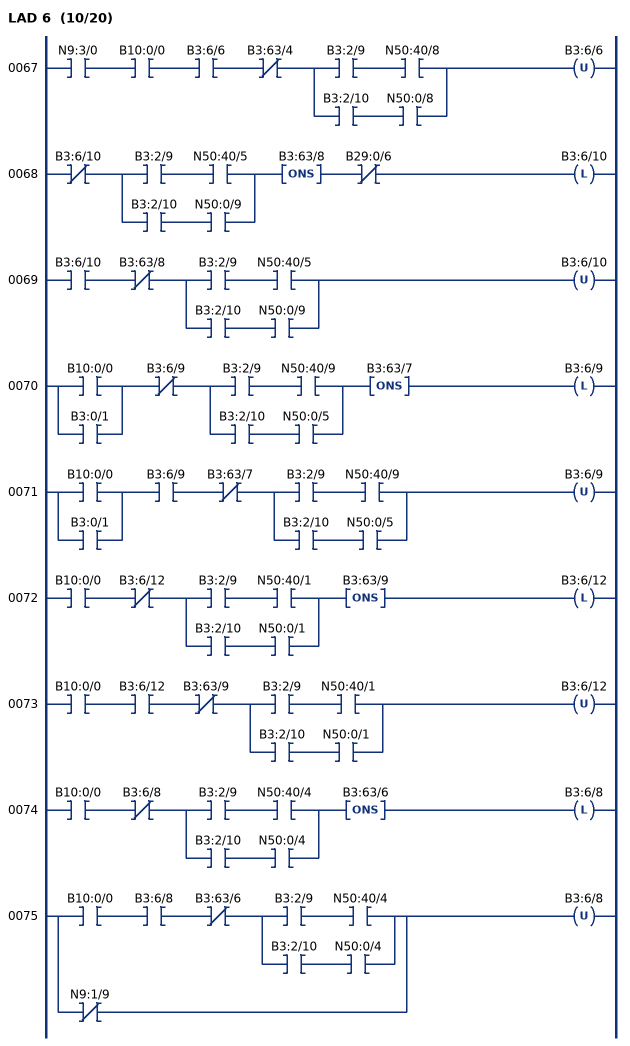
% Rung: 67 %
SOR XIC N9:3/0 XIC B10:0/0 XIC B3:6/6 XIO B3:63/4 BST XIC B3:2/9 XIC N50:40/8 NXB XIC B3:2/10 XIC N50:0/8 BND OTU B3:6/6 EOR
% Rung: 68 %
SOR XIO B3:6/10 BST XIC B3:2/9 XIC N50:40/5 NXB XIC B3:2/10 XIC N50:0/9 BND OSR B3:63/8 XIO B29:0/6 OTL B3:6/10 EOR
% Rung: 69 %
SOR XIC B3:6/10 XIO B3:63/8 BST XIC B3:2/9 XIC N50:40/5 NXB XIC B3:2/10 XIC N50:0/9 BND OTU B3:6/10 EOR
% Rung: 70 %
SOR BST XIC B10:0/0 NXB XIC B3:0/1 BND XIO B3:6/9 BST XIC B3:2/9 XIC N50:40/9 NXB XIC B3:2/10 XIC N50:0/5 BND OSR B3:63/7 OTL B3:6/9 EOR
% Rung: 71 %
SOR BST XIC B10:0/0 NXB XIC B3:0/1 BND XIC B3:6/9 XIO B3:63/7 BST XIC B3:2/9 XIC N50:40/9 NXB XIC B3:2/10 XIC N50:0/5 BND OTU B3:6/9 EOR
% Rung: 72 %
SOR XIC B10:0/0 XIO B3:6/12 BST XIC B3:2/9 XIC N50:40/1 NXB XIC B3:2/10 XIC N50:0/1 BND OSR B3:63/9 OTL B3:6/12 EOR
% Rung: 73 %
SOR XIC B10:0/0 XIC B3:6/12 XIO B3:63/9 BST XIC B3:2/9 XIC N50:40/1 NXB XIC B3:2/10 XIC N50:0/1 BND OTU B3:6/12 EOR
% Rung: 74 %
SOR XIC B10:0/0 XIO B3:6/8 BST XIC B3:2/9 XIC N50:40/4 NXB XIC B3:2/10 XIC N50:0/4 BND OSR B3:63/6 OTL B3:6/8 EOR
% Rung: 75 %
SOR BST XIC B10:0/0 XIC B3:6/8 XIO B3:63/6 BST XIC B3:2/9 XIC N50:40/4 NXB XIC B3:2/10 XIC N50:0/4 BND NXB XIO N9:1/9 BND OTU B3:6/8 EOR

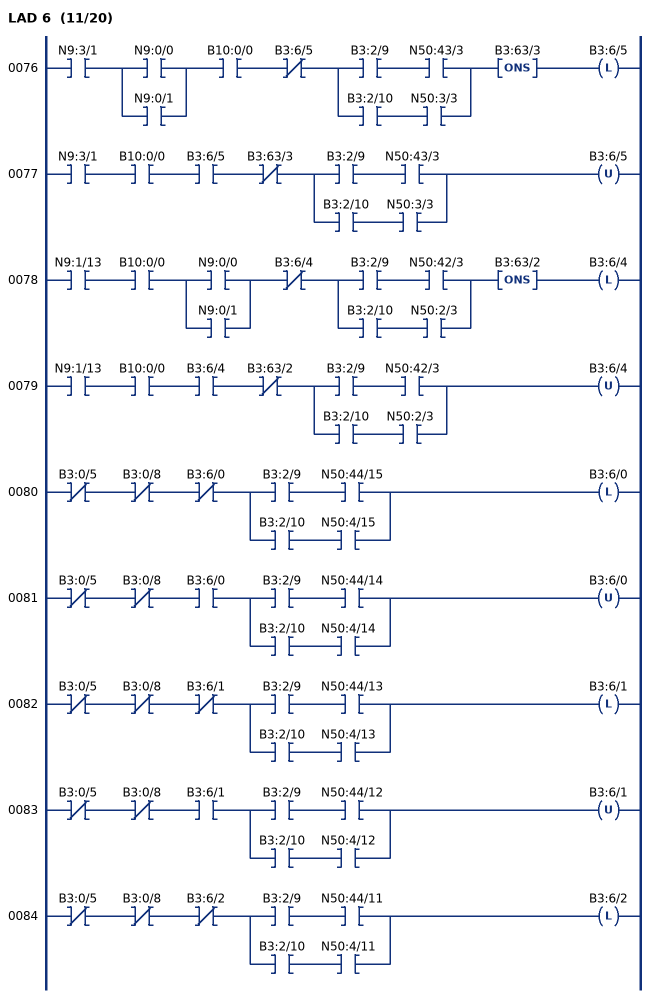
% Rung: 76 %
SOR XIC N9:3/1 BST XIC N9:0/0 NXB XIC N9:0/1 BND XIC B10:0/0 XIO B3:6/5 BST XIC B3:2/9 XIC N50:43/3 NXB XIC B3:2/10 XIC N50:3/3 BND OSR B3:63/3 OTL B3:6/5 EOR
% Rung: 77 %
SOR XIC N9:3/1 XIC B10:0/0 XIC B3:6/5 XIO B3:63/3 BST XIC B3:2/9 XIC N50:43/3 NXB XIC B3:2/10 XIC N50:3/3 BND OTU B3:6/5 EOR
% Rung: 78 %
SOR XIC N9:1/13 XIC B10:0/0 BST XIC N9:0/0 NXB XIC N9:0/1 BND XIO B3:6/4 BST XIC B3:2/9 XIC N50:42/3 NXB XIC B3:2/10 XIC N50:2/3 BND OSR B3:63/2 OTL B3:6/4 EOR
% Rung: 79 %
SOR XIC N9:1/13 XIC B10:0/0 XIC B3:6/4 XIO B3:63/2 BST XIC B3:2/9 XIC N50:42/3 NXB XIC B3:2/10 XIC N50:2/3 BND OTU B3:6/4 EOR
% Rung: 80 %
SOR XIO B3:0/5 XIO B3:0/8 XIO B3:6/0 BST XIC B3:2/9 XIC N50:44/15 NXB XIC B3:2/10 XIC N50:4/15 BND OTL B3:6/0 EOR
% Rung: 81 %
SOR XIO B3:0/5 XIO B3:0/8 XIC B3:6/0 BST XIC B3:2/9 XIC N50:44/14 NXB XIC B3:2/10 XIC N50:4/14 BND OTU B3:6/0 EOR
% Rung: 82 %
SOR XIO B3:0/5 XIO B3:0/8 XIO B3:6/1 BST XIC B3:2/9 XIC N50:44/13 NXB XIC B3:2/10 XIC N50:4/13 BND OTL B3:6/1 EOR
% Rung: 83 %
SOR XIO B3:0/5 XIO B3:0/8 XIC B3:6/1 BST XIC B3:2/9 XIC N50:44/12 NXB XIC B3:2/10 XIC N50:4/12 BND OTU B3:6/1 EOR
% Rung: 84 %
SOR XIO B3:0/5 XIO B3:0/8 XIO B3:6/2 BST XIC B3:2/9 XIC N50:44/11 NXB XIC B3:2/10 XIC N50:4/11 BND OTL B3:6/2 EOR

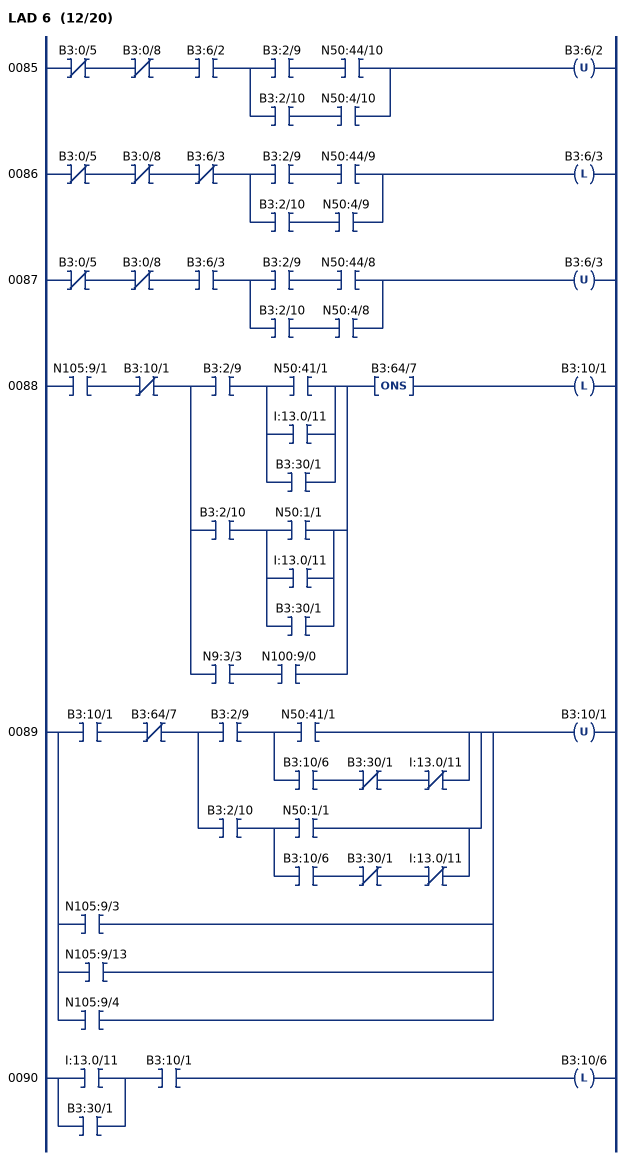
% Rung: 85 %
SOR XIO B3:0/5 XIO B3:0/8 XIC B3:6/2 BST XIC B3:2/9 XIC N50:44/10 NXB XIC B3:2/10 XIC N50:4/10 BND OTU B3:6/2 EOR
% Rung: 86 %
SOR XIO B3:0/5 XIO B3:0/8 XIO B3:6/3 BST XIC B3:2/9 XIC N50:44/9 NXB XIC B3:2/10 XIC N50:4/9 BND OTL B3:6/3 EOR
% Rung: 87 %
SOR XIO B3:0/5 XIO B3:0/8 XIC B3:6/3 BST XIC B3:2/9 XIC N50:44/8 NXB XIC B3:2/10 XIC N50:4/8 BND OTU B3:6/3 EOR
% Rung: 88 %
SOR XIC N105:9/1 XIO B3:10/1 BST XIC B3:2/9 BST XIC N50:41/1 NXB XIC I:13.0/11 NXB XIC B3:30/1 BND NXB XIC B3:2/10 BST XIC N50:1/1 NXB XIC I:13.0/11 NXB XIC B3:30/1 BND NXB XIC N9:3/3 XIC N100:9/0 BND OSR B3:64/7 OTL B3:10/1 EOR
% Rung: 89 %
SOR BST XIC B3:10/1 XIO B3:64/7 BST XIC B3:2/9 BST XIC N50:41/1 NXB XIC B3:10/6 XIO B3:30/1 XIO I:13.0/11 BND NXB XIC B3:2/10 BST XIC N50:1/1 NXB XIC B3:10/6 XIO B3:30/1 XIO I:13.0/11 BND BND NXB XIC N105:9/3 NXB XIC N105:9/13 NXB XIC N105:9/4 BND OTU B3:10/1 EOR
% Rung: 90 %
SOR BST XIC I:13.0/11 NXB XIC B3:30/1 BND XIC B3:10/1 OTL B3:10/6 EOR

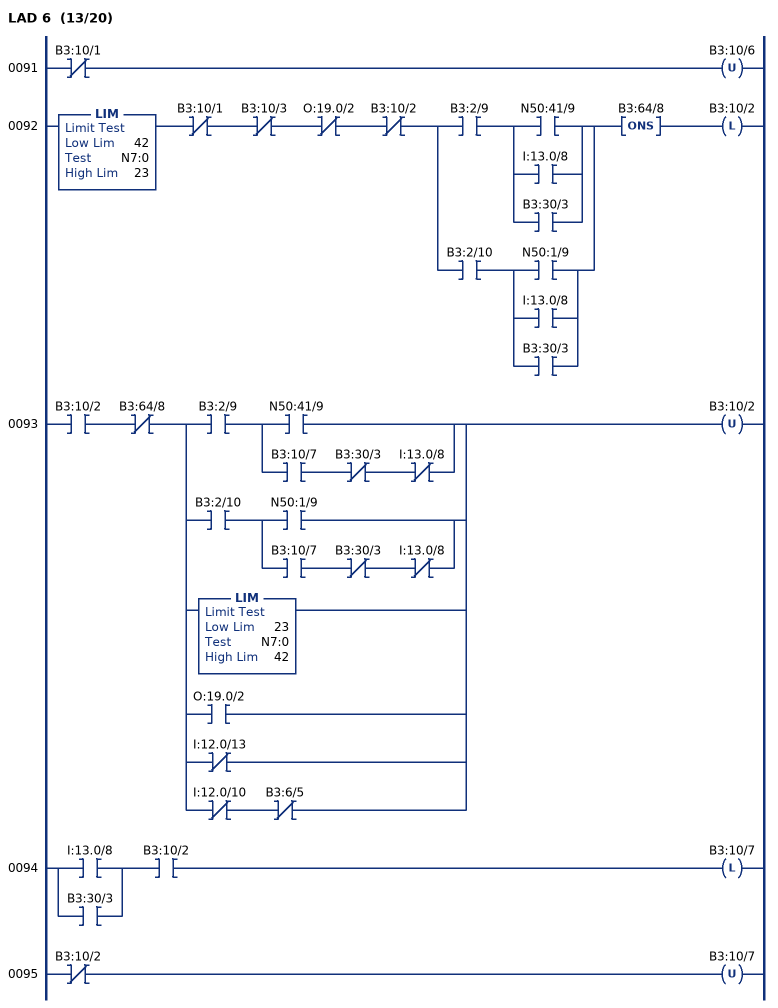
% Rung: 91 %
SOR XIO B3:10/1 OTU B3:10/6 EOR
% Rung: 92 %
SOR LIM 42 N7:0 23 XIO B3:10/1 XIO B3:10/3 XIO O:19.0/2 XIO B3:10/2 BST XIC B3:2/9 BST XIC N50:41/9 NXB XIC I:13.0/8 NXB XIC B3:30/3 BND NXB XIC B3:2/10 BST XIC N50:1/9 NXB XIC I:13.0/8 NXB XIC B3:30/3 BND BND OSR B3:64/8 OTL B3:10/2 EOR
% Rung: 93 %
SOR XIC B3:10/2 XIO B3:64/8 BST XIC B3:2/9 BST XIC N50:41/9 NXB XIC B3:10/7 XIO B3:30/3 XIO I:13.0/8 BND NXB XIC B3:2/10 BST XIC N50:1/9 NXB XIC B3:10/7 XIO B3:30/3 XIO I:13.0/8 BND NXB LIM 23 N7:0 42 NXB XIC O:19.0/2 NXB XIO I:12.0/13 NXB XIO I:12.0/10 XIO B3:6/5 BND OTU B3:10/2 EOR
% Rung: 94 %
SOR BST XIC I:13.0/8 NXB XIC B3:30/3 BND XIC B3:10/2 OTL B3:10/7 EOR
% Rung: 95 %
SOR XIO B3:10/2 OTU B3:10/7 EOR

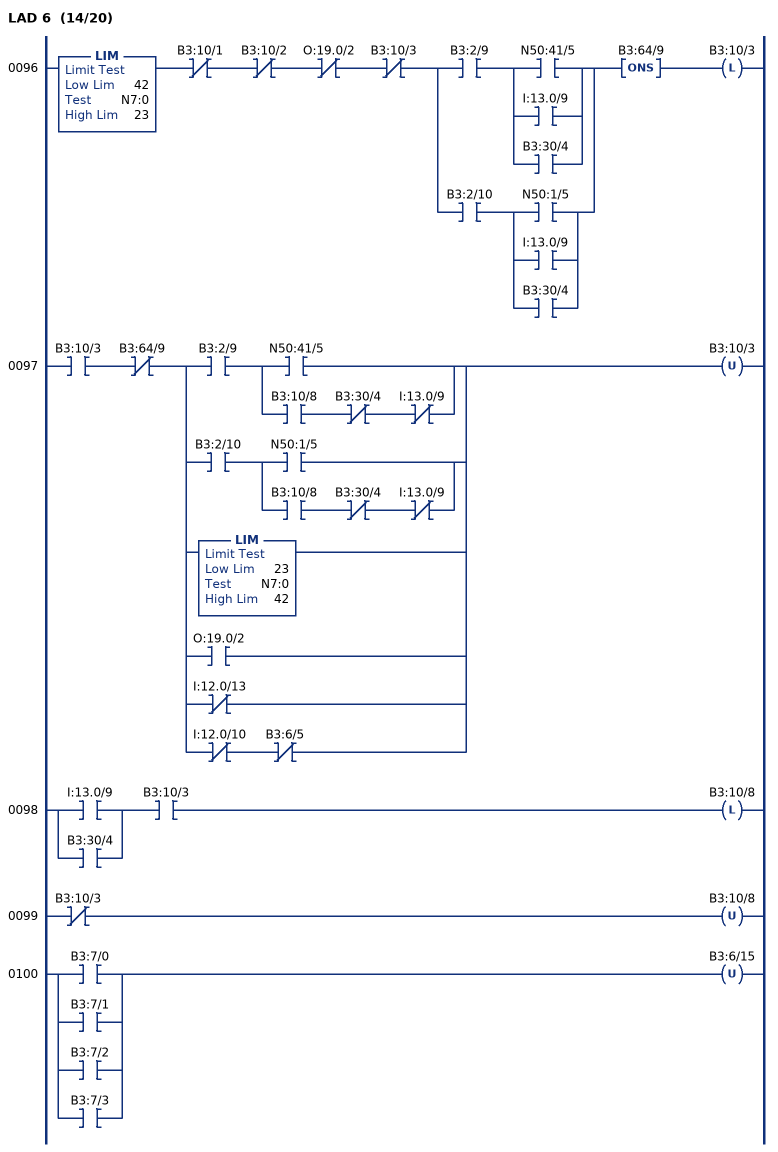
% Rung: 96 %
SOR LIM 42 N7:0 23 XIO B3:10/1 XIO B3:10/2 XIO O:19.0/2 XIO B3:10/3 BST XIC B3:2/9 BST XIC N50:41/5 NXB XIC I:13.0/9 NXB XIC B3:30/4 BND NXB XIC B3:2/10 BST XIC N50:1/5 NXB XIC I:13.0/9 NXB XIC B3:30/4 BND BND OSR B3:64/9 OTL B3:10/3 EOR
% Rung: 97 %
SOR XIC B3:10/3 XIO B3:64/9 BST XIC B3:2/9 BST XIC N50:41/5 NXB XIC B3:10/8 XIO B3:30/4 XIO I:13.0/9 BND NXB XIC B3:2/10 BST XIC N50:1/5 NXB XIC B3:10/8 XIO B3:30/4 XIO I:13.0/9 BND NXB LIM 23 N7:0 42 NXB XIC O:19.0/2 NXB XIO I:12.0/13 NXB XIO I:12.0/10 XIO B3:6/5 BND OTU B3:10/3 EOR
% Rung: 98 %
SOR BST XIC I:13.0/9 NXB XIC B3:30/4 BND XIC B3:10/3 OTL B3:10/8 EOR
% Rung: 99 %
SOR XIO B3:10/3 OTU B3:10/8 EOR
% Rung: 100 %
SOR BST XIC B3:7/0 NXB XIC B3:7/1 NXB XIC B3:7/2 NXB XIC B3:7/3 BND OTU B3:6/15 EOR

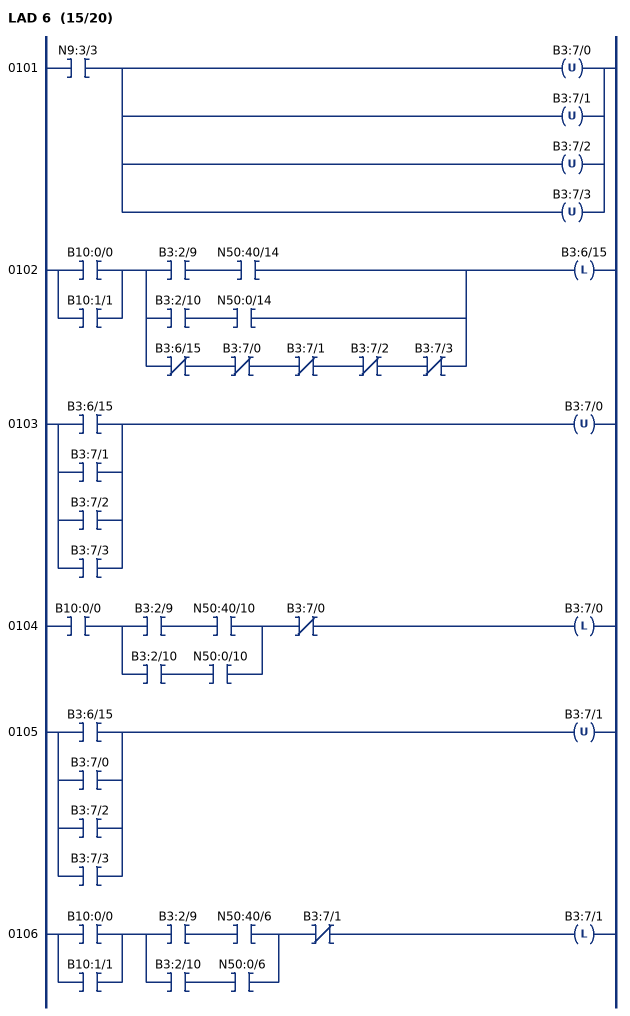
% Rung: 101 %
SOR XIC N9:3/3 BST OTU B3:7/0 NXB OTU B3:7/1 NXB OTU B3:7/2 NXB OTU B3:7/3 BND EOR
% Rung: 102 %
SOR BST XIC B10:0/0 NXB XIC B10:1/1 BND BST XIC B3:2/9 XIC N50:40/14 NXB XIC B3:2/10 XIC N50:0/14 NXB XIO B3:6/15 XIO B3:7/0 XIO B3:7/1 XIO B3:7/2 XIO B3:7/3 BND OTL B3:6/15 EOR
% Rung: 103 %
SOR BST XIC B3:6/15 NXB XIC B3:7/1 NXB XIC B3:7/2 NXB XIC B3:7/3 BND OTU B3:7/0 EOR
% Rung: 104 %
SOR XIC B10:0/0 BST XIC B3:2/9 XIC N50:40/10 NXB XIC B3:2/10 XIC N50:0/10 BND XIO B3:7/0 OTL B3:7/0 EOR
% Rung: 105 %
SOR BST XIC B3:6/15 NXB XIC B3:7/0 NXB XIC B3:7/2 NXB XIC B3:7/3 BND OTU B3:7/1 EOR
% Rung: 106 %
SOR BST XIC B10:0/0 NXB XIC B10:1/1 BND BST XIC B3:2/9 XIC N50:40/6 NXB XIC B3:2/10 XIC N50:0/6 BND XIO B3:7/1 OTL B3:7/1 EOR

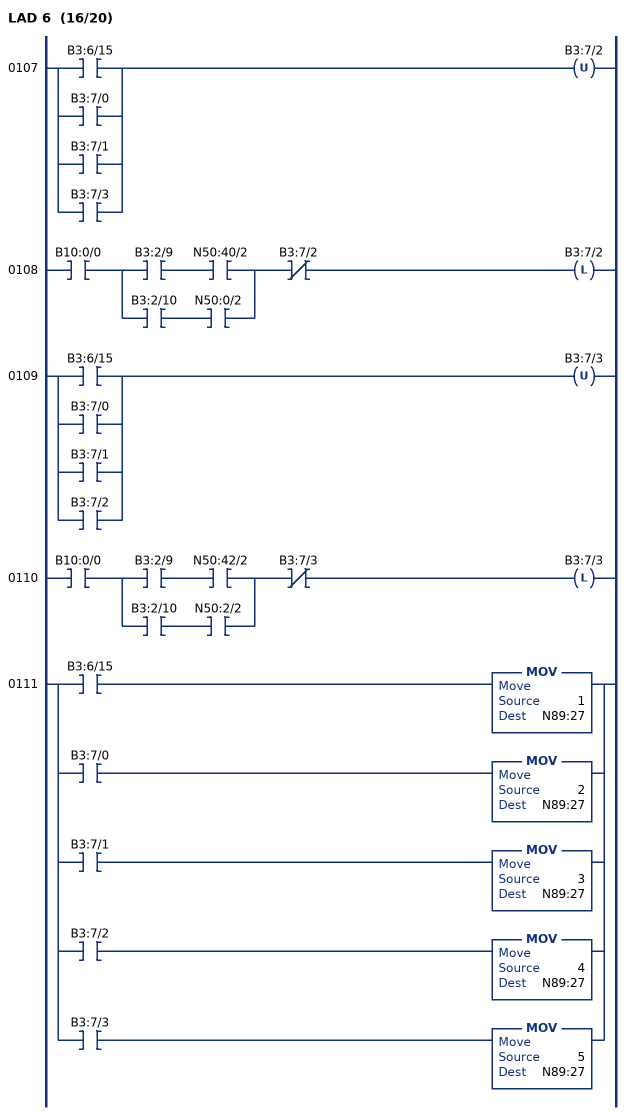
% Rung: 107 %
SOR BST XIC B3:6/15 NXB XIC B3:7/0 NXB XIC B3:7/1 NXB XIC B3:7/3 BND OTU B3:7/2 EOR
% Rung: 108 %
SOR XIC B10:0/0 BST XIC B3:2/9 XIC N50:40/2 NXB XIC B3:2/10 XIC N50:0/2 BND XIO B3:7/2 OTL B3:7/2 EOR
% Rung: 109 %
SOR BST XIC B3:6/15 NXB XIC B3:7/0 NXB XIC B3:7/1 NXB XIC B3:7/2 BND OTU B3:7/3 EOR
% Rung: 110 %
SOR XIC B10:0/0 BST XIC B3:2/9 XIC N50:42/2 NXB XIC B3:2/10 XIC N50:2/2 BND XIO B3:7/3 OTL B3:7/3 EOR
% Rung: 111 %
SOR BST XIC B3:6/15 MOV 1 N89:27 NXB XIC B3:7/0 MOV 2 N89:27 NXB XIC B3:7/1 MOV 3 N89:27 NXB XIC B3:7/2 MOV 4 N89:27 NXB XIC B3:7/3 MOV 5 N89:27 BND EOR

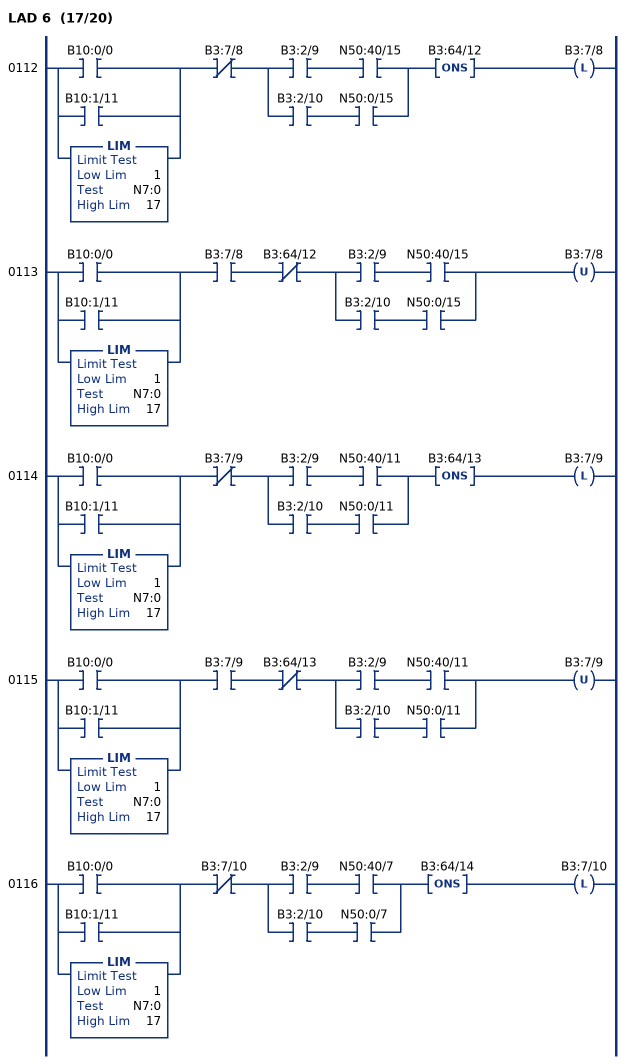
% Rung: 112 %
SOR BST XIC B10:0/0 NXB XIC B10:1/11 NXB LIM 1 N7:0 17 BND XIO B3:7/8 BST XIC B3:2/9 XIC N50:40/15 NXB XIC B3:2/10 XIC N50:0/15 BND OSR B3:64/12 OTL B3:7/8 EOR
% Rung: 113 %
SOR BST XIC B10:0/0 NXB XIC B10:1/11 NXB LIM 1 N7:0 17 BND XIC B3:7/8 XIO B3:64/12 BST XIC B3:2/9 XIC N50:40/15 NXB XIC B3:2/10 XIC N50:0/15 BND OTU B3:7/8 EOR
% Rung: 114 %
SOR BST XIC B10:0/0 NXB XIC B10:1/11 NXB LIM 1 N7:0 17 BND XIO B3:7/9 BST XIC B3:2/9 XIC N50:40/11 NXB XIC B3:2/10 XIC N50:0/11 BND OSR B3:64/13 OTL B3:7/9 EOR
% Rung: 115 %
SOR BST XIC B10:0/0 NXB XIC B10:1/11 NXB LIM 1 N7:0 17 BND XIC B3:7/9 XIO B3:64/13 BST XIC B3:2/9 XIC N50:40/11 NXB XIC B3:2/10 XIC N50:0/11 BND OTU B3:7/9 EOR
% Rung: 116 %
SOR BST XIC B10:0/0 NXB XIC B10:1/11 NXB LIM 1 N7:0 17 BND XIO B3:7/10 BST XIC B3:2/9 XIC N50:40/7 NXB XIC B3:2/10 XIC N50:0/7 BND OSR B3:64/14 OTL B3:7/10 EOR

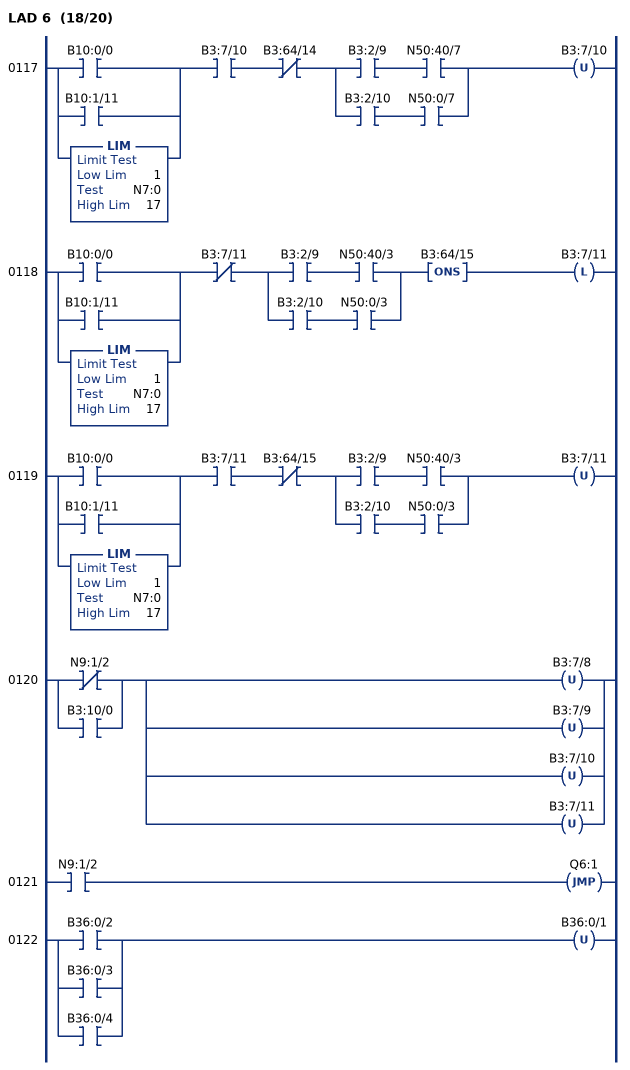
% Rung: 117 %
SOR BST XIC B10:0/0 NXB XIC B10:1/11 NXB LIM 1 N7:0 17 BND XIC B3:7/10 XIO B3:64/14 BST XIC B3:2/9 XIC N50:40/7 NXB XIC B3:2/10 XIC N50:0/7 BND OTU B3:7/10 EOR
% Rung: 118 %
SOR BST XIC B10:0/0 NXB XIC B10:1/11 NXB LIM 1 N7:0 17 BND XIO B3:7/11 BST XIC B3:2/9 XIC N50:40/3 NXB XIC B3:2/10 XIC N50:0/3 BND OSR B3:64/15 OTL B3:7/11 EOR
% Rung: 119 %
SOR BST XIC B10:0/0 NXB XIC B10:1/11 NXB LIM 1 N7:0 17 BND XIC B3:7/11 XIO B3:64/15 BST XIC B3:2/9 XIC N50:40/3 NXB XIC B3:2/10 XIC N50:0/3 BND OTU B3:7/11 EOR
% Rung: 120 %
SOR BST XIO N9:1/2 NXB XIC B3:10/0 BND BST OTU B3:7/8 NXB OTU B3:7/9 NXB OTU B3:7/10 NXB OTU B3:7/11 BND EOR
% Rung: 121 %
SOR XIC N9:1/2 JMP Q6:1 EOR
% Rung: 122 %
SOR BST XIC B36:0/2 NXB XIC B36:0/3 NXB XIC B36:0/4 BND OTU B36:0/1 EOR

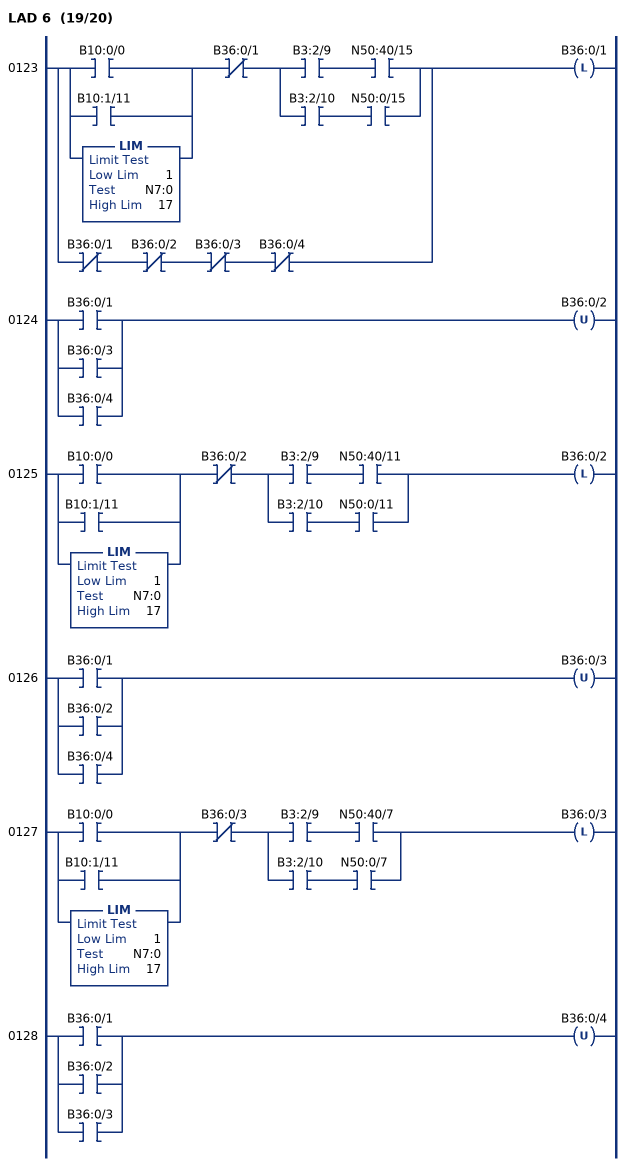
% Rung: 123 %
SOR BST BST XIC B10:0/0 NXB XIC B10:1/11 NXB LIM 1 N7:0 17 BND XIO B36:0/1 BST XIC B3:2/9 XIC N50:40/15 NXB XIC B3:2/10 XIC N50:0/15 BND NXB XIO B36:0/1 XIO B36:0/2 XIO B36:0/3 XIO B36:0/4 BND OTL B36:0/1 EOR
% Rung: 124 %
SOR BST XIC B36:0/1 NXB XIC B36:0/3 NXB XIC B36:0/4 BND OTU B36:0/2 EOR
% Rung: 125 %
SOR BST XIC B10:0/0 NXB XIC B10:1/11 NXB LIM 1 N7:0 17 BND XIO B36:0/2 BST XIC B3:2/9 XIC N50:40/11 NXB XIC B3:2/10 XIC N50:0/11 BND OTL B36:0/2 EOR
% Rung: 126 %
SOR BST XIC B36:0/1 NXB XIC B36:0/2 NXB XIC B36:0/4 BND OTU B36:0/3 EOR
% Rung: 127 %
SOR BST XIC B10:0/0 NXB XIC B10:1/11 NXB LIM 1 N7:0 17 BND XIO B36:0/3 BST XIC B3:2/9 XIC N50:40/7 NXB XIC B3:2/10 XIC N50:0/7 BND OTL B36:0/3 EOR
% Rung: 128 %
SOR BST XIC B36:0/1 NXB XIC B36:0/2 NXB XIC B36:0/3 BND OTU B36:0/4 EOR

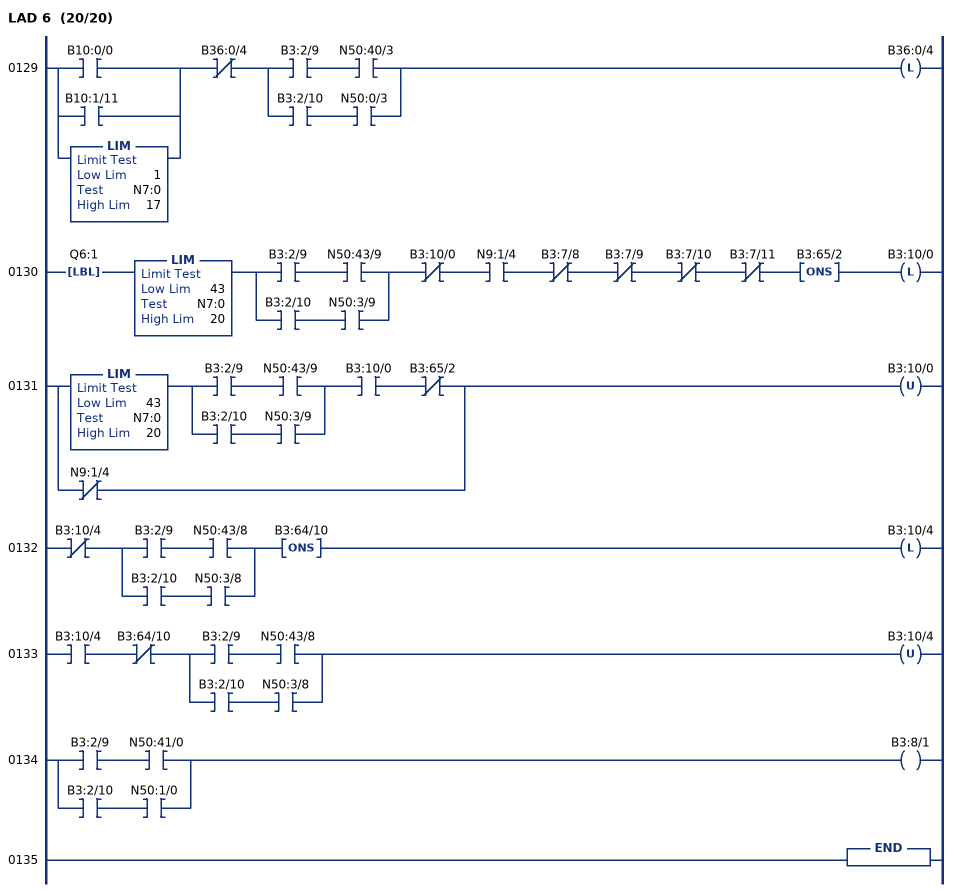
% Rung: 129 %
SOR BST XIC B10:0/0 NXB XIC B10:1/11 NXB LIM 1 N7:0 17 BND XIO B36:0/4 BST XIC B3:2/9 XIC N50:40/3 NXB XIC B3:2/10 XIC N50:0/3 BND OTL B36:0/4 EOR
% Rung: 130 %
SOR LBL Q6:1 LIM 43 N7:0 20 BST XIC B3:2/9 XIC N50:43/9 NXB XIC B3:2/10 XIC N50:3/9 BND XIO B3:10/0 XIC N9:1/4 XIO B3:7/8 XIO B3:7/9 XIO B3:7/10 XIO B3:7/11 OSR B3:65/2 OTL B3:10/0 EOR
% Rung: 131 %
SOR BST LIM 43 N7:0 20 BST XIC B3:2/9 XIC N50:43/9 NXB XIC B3:2/10 XIC N50:3/9 BND XIC B3:10/0 XIO B3:65/2 NXB XIO N9:1/4 BND OTU B3:10/0 EOR
% Rung: 132 %
SOR XIO B3:10/4 BST XIC B3:2/9 XIC N50:43/8 NXB XIC B3:2/10 XIC N50:3/8 BND OSR B3:64/10 OTL B3:10/4 EOR
% Rung: 133 %
SOR XIC B3:10/4 XIO B3:64/10 BST XIC B3:2/9 XIC N50:43/8 NXB XIC B3:2/10 XIC N50:3/8 BND OTU B3:10/4 EOR
% Rung: 134 %
SOR BST XIC B3:2/9 XIC N50:41/0 NXB XIC B3:2/10 XIC N50:1/0 BND OTE B3:8/1 EOR
% Rung: 135 %
SOR END EOR

LADDER 9
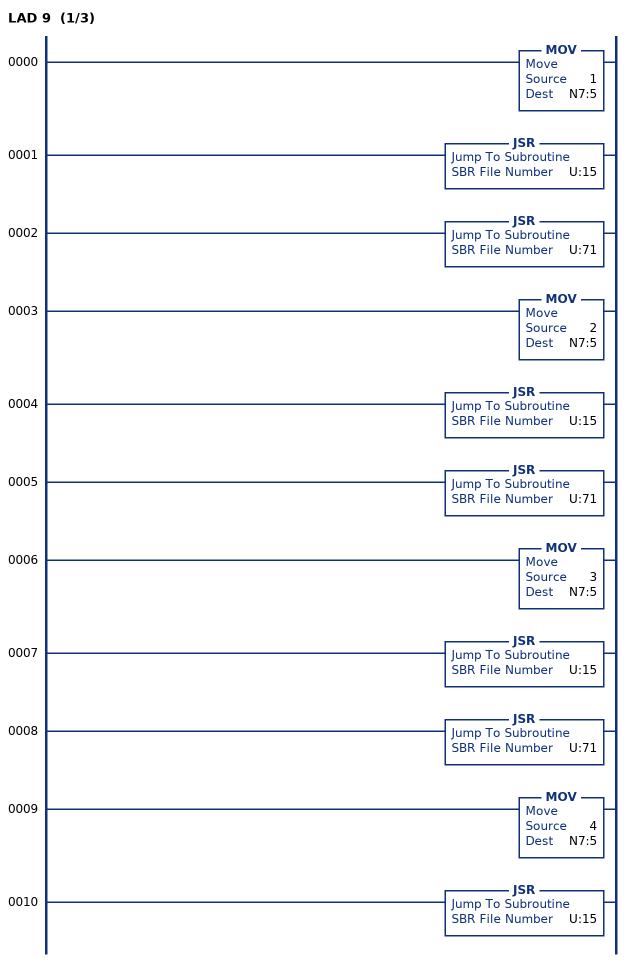
% Rung: 0 %
SOR MOV 1 N7:5 EOR
% Rung: 1 %
SOR JSR U:15 EOR
% Rung: 2 %
SOR JSR U:71 EOR
% Rung: 3 %
SOR MOV 2 N7:5 EOR
% Rung: 4 %
SOR JSR U:15 EOR
% Rung: 5 %
SOR JSR U:71 EOR
% Rung: 6 %
SOR MOV 3 N7:5 EOR
% Rung: 7 %
SOR JSR U:15 EOR
% Rung: 8 %
SOR JSR U:71 EOR
% Rung: 9 %
SOR MOV 4 N7:5 EOR
% Rung: 10 %
SOR JSR U:15 EOR

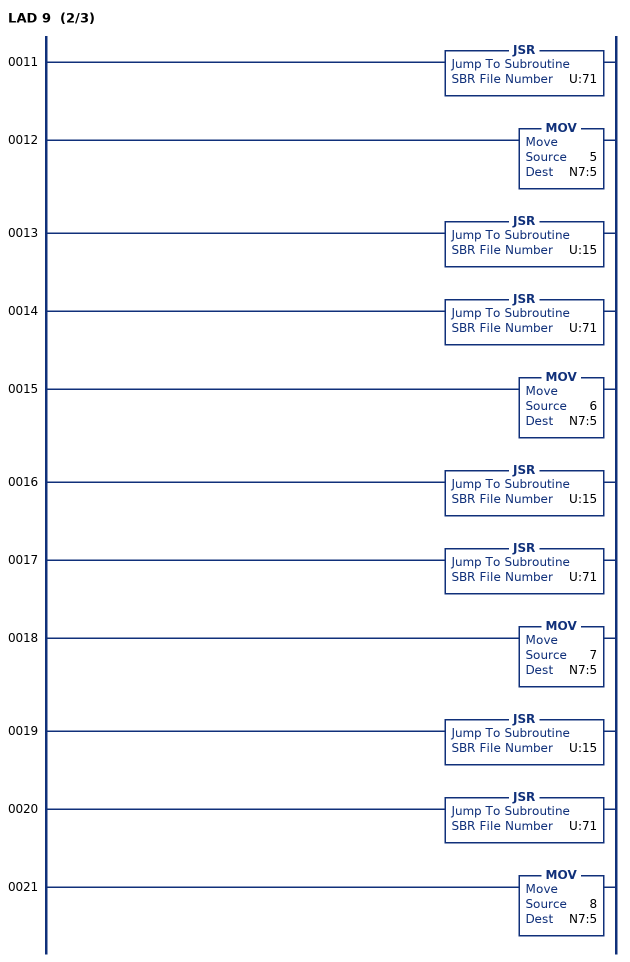
% Rung: 11 %
SOR JSR U:71 EOR
% Rung: 12 %
SOR MOV 5 N7:5 EOR
% Rung: 13 %
SOR JSR U:15 EOR
% Rung: 14 %
SOR JSR U:71 EOR
% Rung: 15 %
SOR MOV 6 N7:5 EOR
% Rung: 16 %
SOR JSR U:15 EOR
% Rung: 17 %
SOR JSR U:71 EOR
% Rung: 18 %
SOR MOV 7 N7:5 EOR
% Rung: 19 %
SOR JSR U:15 EOR
% Rung: 20 %
SOR JSR U:71 EOR
% Rung: 21 %
SOR MOV 8 N7:5 EOR

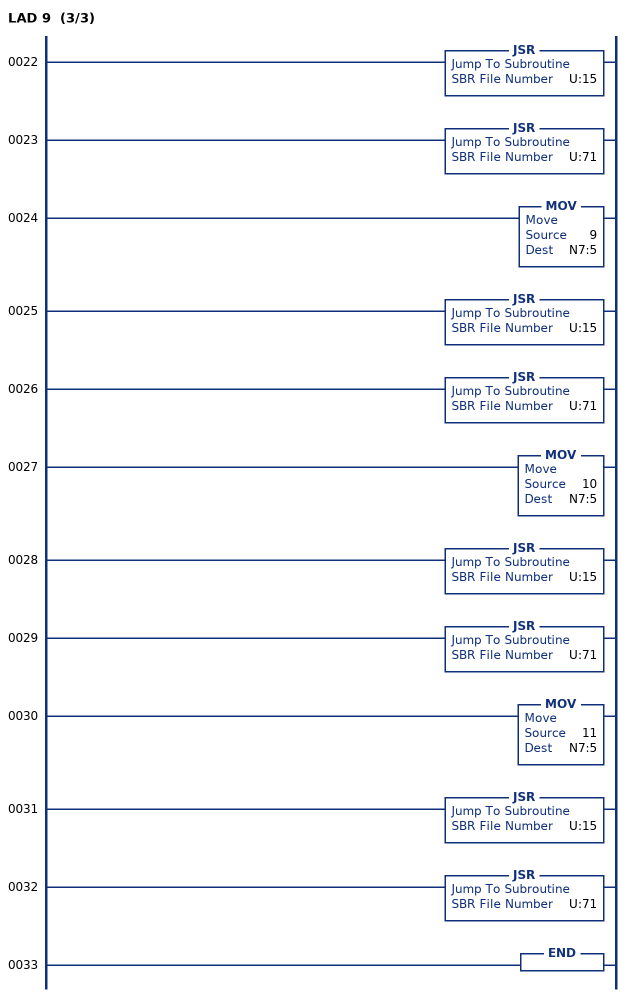
% Rung: 22 %
SOR JSR U:15 EOR
% Rung: 23 %
SOR JSR U:71 EOR
% Rung: 24 %
SOR MOV 9 N7:5 EOR
% Rung: 25 %
SOR JSR U:15 EOR
% Rung: 26 %
SOR JSR U:71 EOR
% Rung: 27 %
SOR MOV 10 N7:5 EOR
% Rung: 28 %
SOR JSR U:15 EOR
% Rung: 29 %
SOR JSR U:71 EOR
% Rung: 30 %
SOR MOV 11 N7:5 EOR
% Rung: 31 %
SOR JSR U:15 EOR
% Rung: 32 %
SOR JSR U:71 EOR
% Rung: 33 %
SOR END EOR

LADDER 10
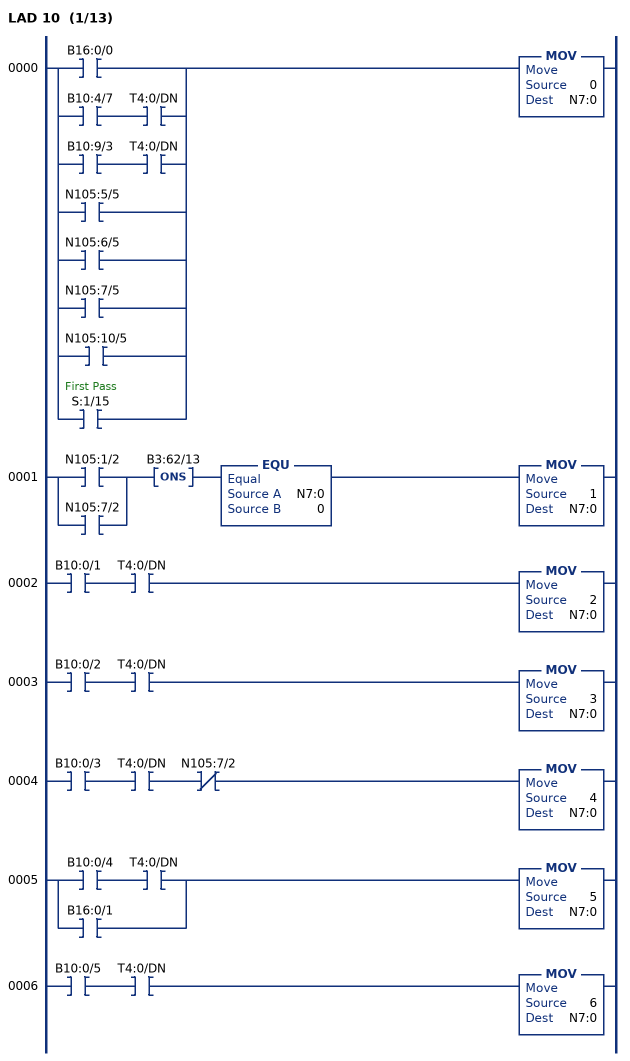
% Rung: 0 %
SOR BST XIC B16:0/0 NXB XIC B10:4/7 XIC T4:0/DN NXB XIC B10:9/3 XIC T4:0/DN NXB XIC N105:5/5 NXB XIC N105:6/5 NXB XIC N105:7/5 NXB XIC N105:10/5 NXB XIC S:1/15 BND MOV 0 N7:0 EOR
%   S:1/15  "First Pass" %
% Rung: 1 %
SOR BST XIC N105:1/2 NXB XIC N105:7/2 BND OSR B3:62/13 EQU N7:0 0 MOV 1 N7:0 EOR
% Rung: 2 %
SOR XIC B10:0/1 XIC T4:0/DN MOV 2 N7:0 EOR
% Rung: 3 %
SOR XIC B10:0/2 XIC T4:0/DN MOV 3 N7:0 EOR
% Rung: 4 %
SOR XIC B10:0/3 XIC T4:0/DN XIO N105:7/2 MOV 4 N7:0 EOR
% Rung: 5 %
SOR BST XIC B10:0/4 XIC T4:0/DN NXB XIC B16:0/1 BND MOV 5 N7:0 EOR
% Rung: 6 %
SOR XIC B10:0/5 XIC T4:0/DN MOV 6 N7:0 EOR

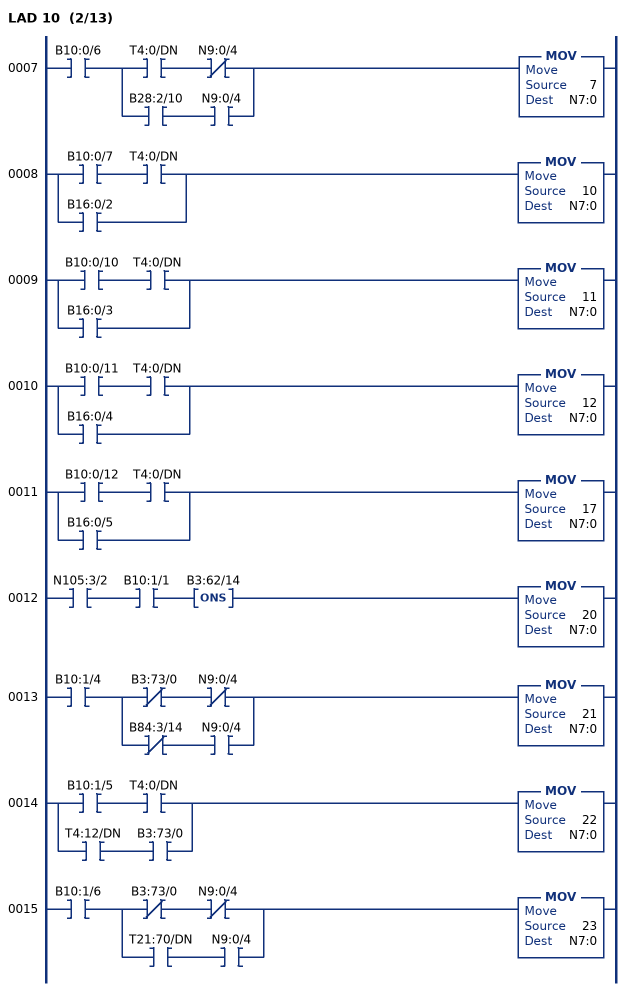
% Rung: 7 %
SOR XIC B10:0/6 BST XIC T4:0/DN XIO N9:0/4 NXB XIC B28:2/10 XIC N9:0/4 BND MOV 7 N7:0 EOR
% Rung: 8 %
SOR BST XIC B10:0/7 XIC T4:0/DN NXB XIC B16:0/2 BND MOV 10 N7:0 EOR
% Rung: 9 %
SOR BST XIC B10:0/10 XIC T4:0/DN NXB XIC B16:0/3 BND MOV 11 N7:0 EOR
% Rung: 10 %
SOR BST XIC B10:0/11 XIC T4:0/DN NXB XIC B16:0/4 BND MOV 12 N7:0 EOR
% Rung: 11 %
SOR BST XIC B10:0/12 XIC T4:0/DN NXB XIC B16:0/5 BND MOV 17 N7:0 EOR
% Rung: 12 %
SOR XIC N105:3/2 XIC B10:1/1 OSR B3:62/14 MOV 20 N7:0 EOR
% Rung: 13 %
SOR XIC B10:1/4 BST XIO B3:73/0 XIO N9:0/4 NXB XIO B84:3/14 XIC N9:0/4 BND MOV 21 N7:0 EOR
% Rung: 14 %
SOR BST XIC B10:1/5 XIC T4:0/DN NXB XIC T4:12/DN XIC B3:73/0 BND MOV 22 N7:0 EOR
% Rung: 15 %
SOR XIC B10:1/6 BST XIO B3:73/0 XIO N9:0/4 NXB XIC T21:70/DN XIC N9:0/4 BND MOV 23 N7:0 EOR

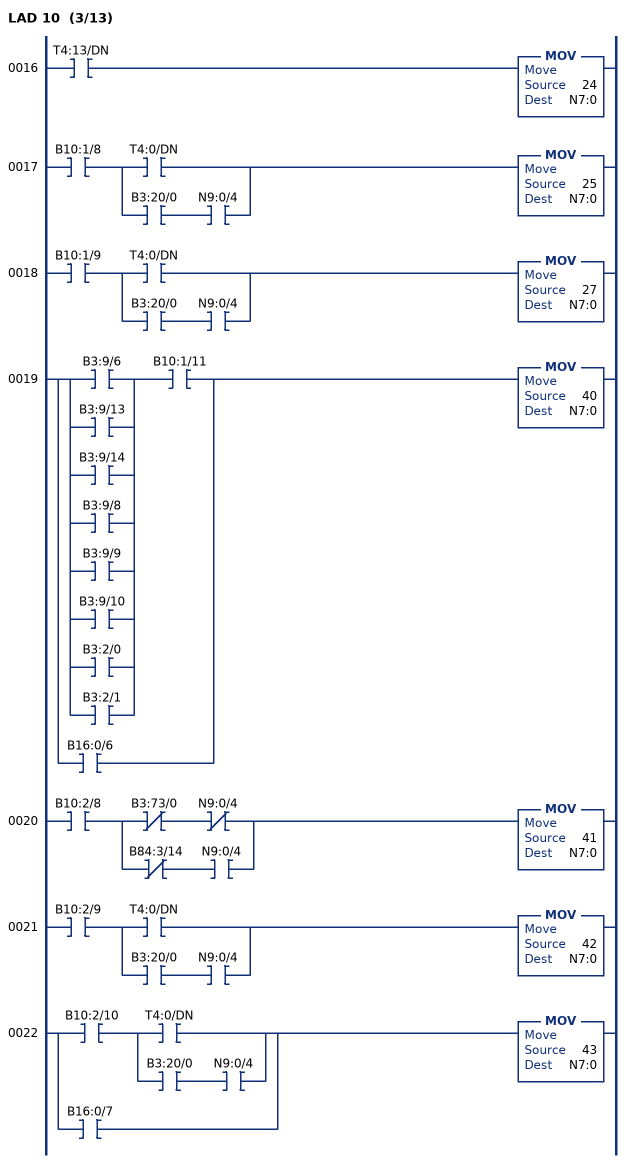
% Rung: 16 %
SOR XIC T4:13/DN MOV 24 N7:0 EOR
% Rung: 17 %
SOR XIC B10:1/8 BST XIC T4:0/DN NXB XIC B3:20/0 XIC N9:0/4 BND MOV 25 N7:0 EOR
% Rung: 18 %
SOR XIC B10:1/9 BST XIC T4:0/DN NXB XIC B3:20/0 XIC N9:0/4 BND MOV 27 N7:0 EOR
% Rung: 19 %
SOR BST BST XIC B3:9/6 NXB XIC B3:9/13 NXB XIC B3:9/14 NXB XIC B3:9/8 NXB XIC B3:9/9 NXB XIC B3:9/10 NXB XIC B3:2/0 NXB XIC B3:2/1 BND XIC B10:1/11 NXB XIC B16:0/6 BND MOV 40 N7:0 EOR
% Rung: 20 %
SOR XIC B10:2/8 BST XIO B3:73/0 XIO N9:0/4 NXB XIO B84:3/14 XIC N9:0/4 BND MOV 41 N7:0 EOR
% Rung: 21 %
SOR XIC B10:2/9 BST XIC T4:0/DN NXB XIC B3:20/0 XIC N9:0/4 BND MOV 42 N7:0 EOR
% Rung: 22 %
SOR BST XIC B10:2/10 BST XIC T4:0/DN NXB XIC B3:20/0 XIC N9:0/4 BND NXB XIC B16:0/7 BND MOV 43 N7:0 EOR

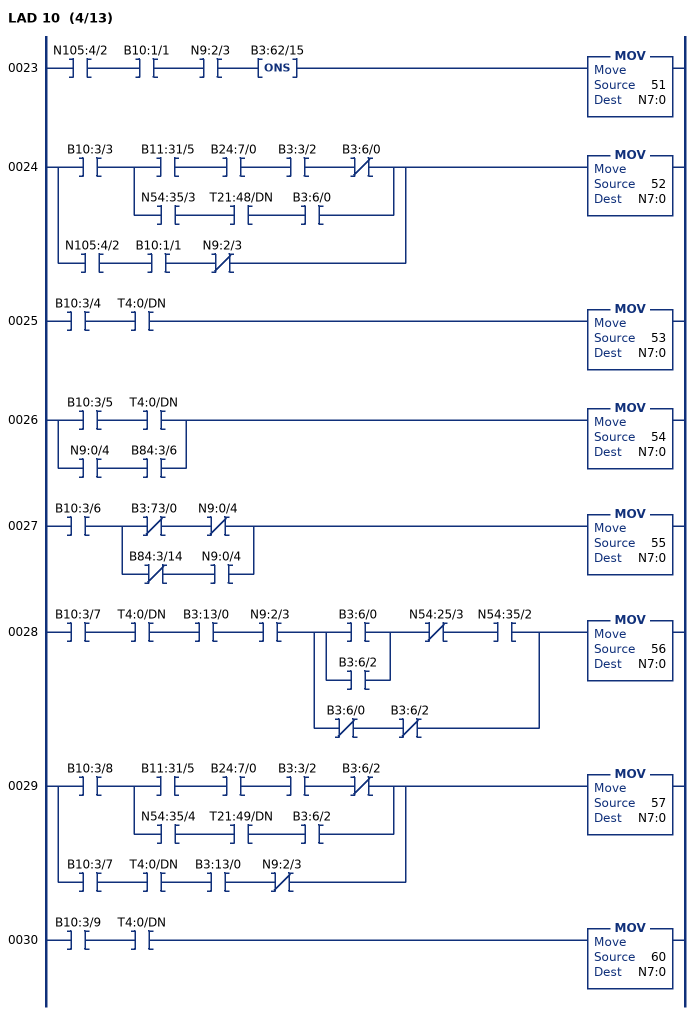
% Rung: 23 %
SOR XIC N105:4/2 XIC B10:1/1 XIC N9:2/3 OSR B3:62/15 MOV 51 N7:0 EOR
% Rung: 24 %
SOR BST XIC B10:3/3 BST XIC B11:31/5 XIC B24:7/0 XIC B3:3/2 XIO B3:6/0 NXB XIC N54:35/3 XIC T21:48/DN XIC B3:6/0 BND NXB XIC N105:4/2 XIC B10:1/1 XIO N9:2/3 BND MOV 52 N7:0 EOR
% Rung: 25 %
SOR XIC B10:3/4 XIC T4:0/DN MOV 53 N7:0 EOR
% Rung: 26 %
SOR BST XIC B10:3/5 XIC T4:0/DN NXB XIC N9:0/4 XIC B84:3/6 BND MOV 54 N7:0 EOR
% Rung: 27 %
SOR XIC B10:3/6 BST XIO B3:73/0 XIO N9:0/4 NXB XIO B84:3/14 XIC N9:0/4 BND MOV 55 N7:0 EOR
% Rung: 28 %
SOR XIC B10:3/7 XIC T4:0/DN XIC B3:13/0 XIC N9:2/3 BST BST XIC B3:6/0 NXB XIC B3:6/2 BND XIO N54:25/3 XIC N54:35/2 NXB XIO B3:6/0 XIO B3:6/2 BND MOV 56 N7:0 EOR
% Rung: 29 %
SOR BST XIC B10:3/8 BST XIC B11:31/5 XIC B24:7/0 XIC B3:3/2 XIO B3:6/2 NXB XIC N54:35/4 XIC T21:49/DN XIC B3:6/2 BND NXB XIC B10:3/7 XIC T4:0/DN XIC B3:13/0 XIO N9:2/3 BND MOV 57 N7:0 EOR
% Rung: 30 %
SOR XIC B10:3/9 XIC T4:0/DN MOV 60 N7:0 EOR

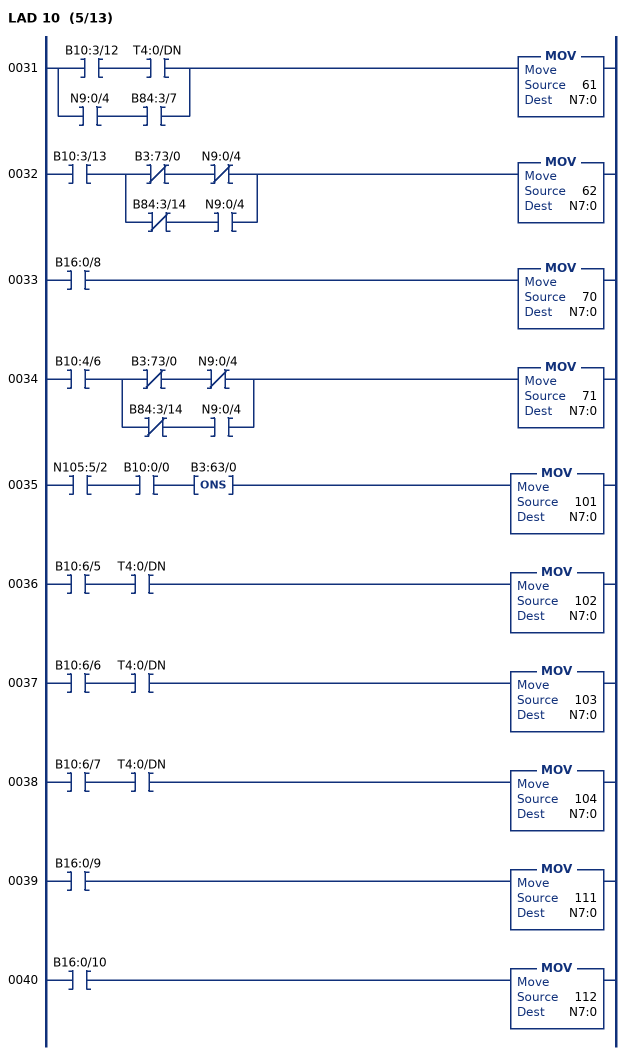
% Rung: 31 %
SOR BST XIC B10:3/12 XIC T4:0/DN NXB XIC N9:0/4 XIC B84:3/7 BND MOV 61 N7:0 EOR
% Rung: 32 %
SOR XIC B10:3/13 BST XIO B3:73/0 XIO N9:0/4 NXB XIO B84:3/14 XIC N9:0/4 BND MOV 62 N7:0 EOR
% Rung: 33 %
SOR XIC B16:0/8 MOV 70 N7:0 EOR
% Rung: 34 %
SOR XIC B10:4/6 BST XIO B3:73/0 XIO N9:0/4 NXB XIO B84:3/14 XIC N9:0/4 BND MOV 71 N7:0 EOR
% Rung: 35 %
SOR XIC N105:5/2 XIC B10:0/0 OSR B3:63/0 MOV 101 N7:0 EOR
% Rung: 36 %
SOR XIC B10:6/5 XIC T4:0/DN MOV 102 N7:0 EOR
% Rung: 37 %
SOR XIC B10:6/6 XIC T4:0/DN MOV 103 N7:0 EOR
% Rung: 38 %
SOR XIC B10:6/7 XIC T4:0/DN MOV 104 N7:0 EOR
% Rung: 39 %
SOR XIC B16:0/9 MOV 111 N7:0 EOR
% Rung: 40 %
SOR XIC B16:0/10 MOV 112 N7:0 EOR

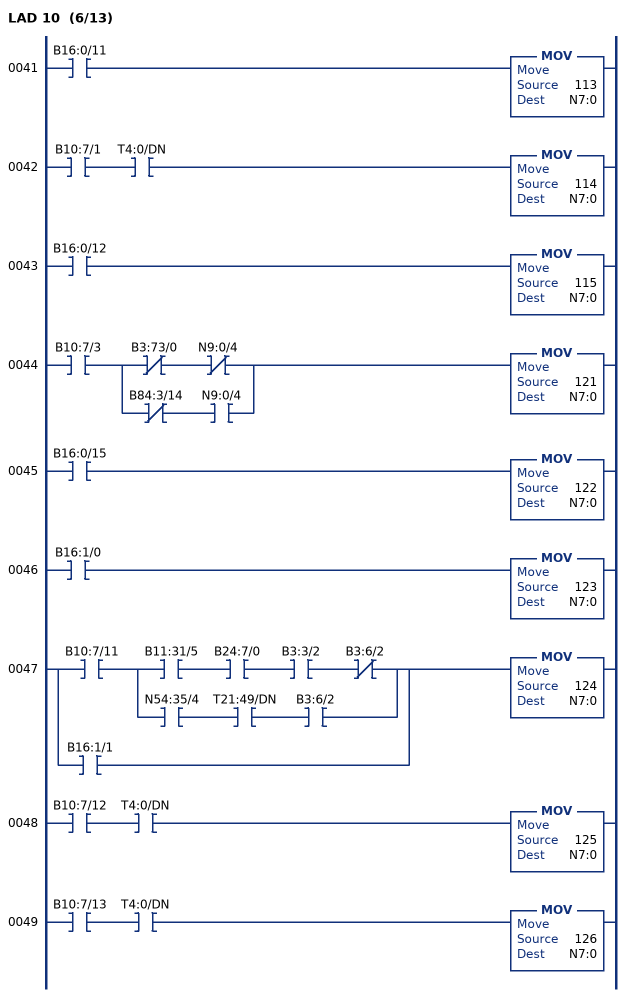
% Rung: 41 %
SOR XIC B16:0/11 MOV 113 N7:0 EOR
% Rung: 42 %
SOR XIC B10:7/1 XIC T4:0/DN MOV 114 N7:0 EOR
% Rung: 43 %
SOR XIC B16:0/12 MOV 115 N7:0 EOR
% Rung: 44 %
SOR XIC B10:7/3 BST XIO B3:73/0 XIO N9:0/4 NXB XIO B84:3/14 XIC N9:0/4 BND MOV 121 N7:0 EOR
% Rung: 45 %
SOR XIC B16:0/15 MOV 122 N7:0 EOR
% Rung: 46 %
SOR XIC B16:1/0 MOV 123 N7:0 EOR
% Rung: 47 %
SOR BST XIC B10:7/11 BST XIC B11:31/5 XIC B24:7/0 XIC B3:3/2 XIO B3:6/2 NXB XIC N54:35/4 XIC T21:49/DN XIC B3:6/2 BND NXB XIC B16:1/1 BND MOV 124 N7:0 EOR
% Rung: 48 %
SOR XIC B10:7/12 XIC T4:0/DN MOV 125 N7:0 EOR
% Rung: 49 %
SOR XIC B10:7/13 XIC T4:0/DN MOV 126 N7:0 EOR

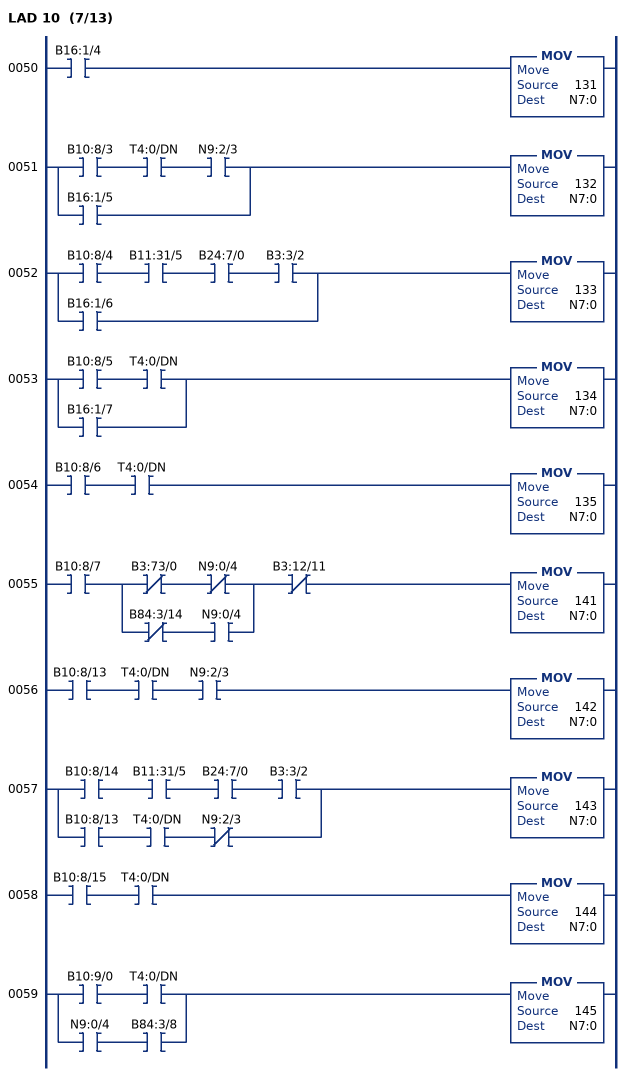
% Rung: 50 %
SOR XIC B16:1/4 MOV 131 N7:0 EOR
% Rung: 51 %
SOR BST XIC B10:8/3 XIC T4:0/DN XIC N9:2/3 NXB XIC B16:1/5 BND MOV 132 N7:0 EOR
% Rung: 52 %
SOR BST XIC B10:8/4 XIC B11:31/5 XIC B24:7/0 XIC B3:3/2 NXB XIC B16:1/6 BND MOV 133 N7:0 EOR
% Rung: 53 %
SOR BST XIC B10:8/5 XIC T4:0/DN NXB XIC B16:1/7 BND MOV 134 N7:0 EOR
% Rung: 54 %
SOR XIC B10:8/6 XIC T4:0/DN MOV 135 N7:0 EOR
% Rung: 55 %
SOR XIC B10:8/7 BST XIO B3:73/0 XIO N9:0/4 NXB XIO B84:3/14 XIC N9:0/4 BND XIO B3:12/11 MOV 141 N7:0 EOR
% Rung: 56 %
SOR XIC B10:8/13 XIC T4:0/DN XIC N9:2/3 MOV 142 N7:0 EOR
% Rung: 57 %
SOR BST XIC B10:8/14 XIC B11:31/5 XIC B24:7/0 XIC B3:3/2 NXB XIC B10:8/13 XIC T4:0/DN XIO N9:2/3 BND MOV 143 N7:0 EOR
% Rung: 58 %
SOR XIC B10:8/15 XIC T4:0/DN MOV 144 N7:0 EOR
% Rung: 59 %
SOR BST XIC B10:9/0 XIC T4:0/DN NXB XIC N9:0/4 XIC B84:3/8 BND MOV 145 N7:0 EOR

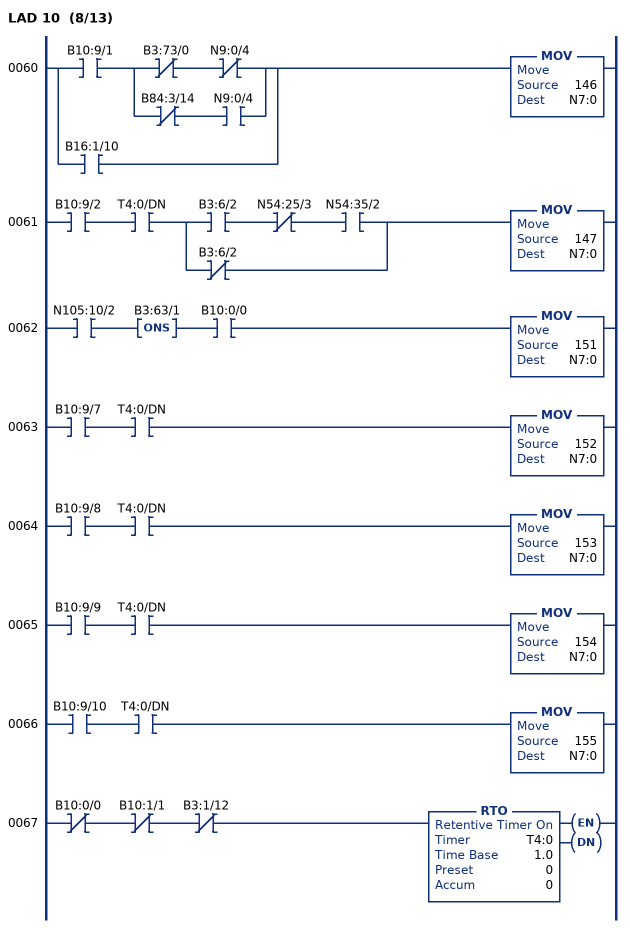
% Rung: 60 %
SOR BST XIC B10:9/1 BST XIO B3:73/0 XIO N9:0/4 NXB XIO B84:3/14 XIC N9:0/4 BND NXB XIC B16:1/10 BND MOV 146 N7:0 EOR
% Rung: 61 %
SOR XIC B10:9/2 XIC T4:0/DN BST XIC B3:6/2 XIO N54:25/3 XIC N54:35/2 NXB XIO B3:6/2 BND MOV 147 N7:0 EOR
% Rung: 62 %
SOR XIC N105:10/2 OSR B3:63/1 XIC B10:0/0 MOV 151 N7:0 EOR
% Rung: 63 %
SOR XIC B10:9/7 XIC T4:0/DN MOV 152 N7:0 EOR
% Rung: 64 %
SOR XIC B10:9/8 XIC T4:0/DN MOV 153 N7:0 EOR
% Rung: 65 %
SOR XIC B10:9/9 XIC T4:0/DN MOV 154 N7:0 EOR
% Rung: 66 %
SOR XIC B10:9/10 XIC T4:0/DN MOV 155 N7:0 EOR
% Rung: 67 %
SOR XIO B10:0/0 XIO B10:1/1 XIO B3:1/12 RTO T4:0 1.0 0 0 EOR

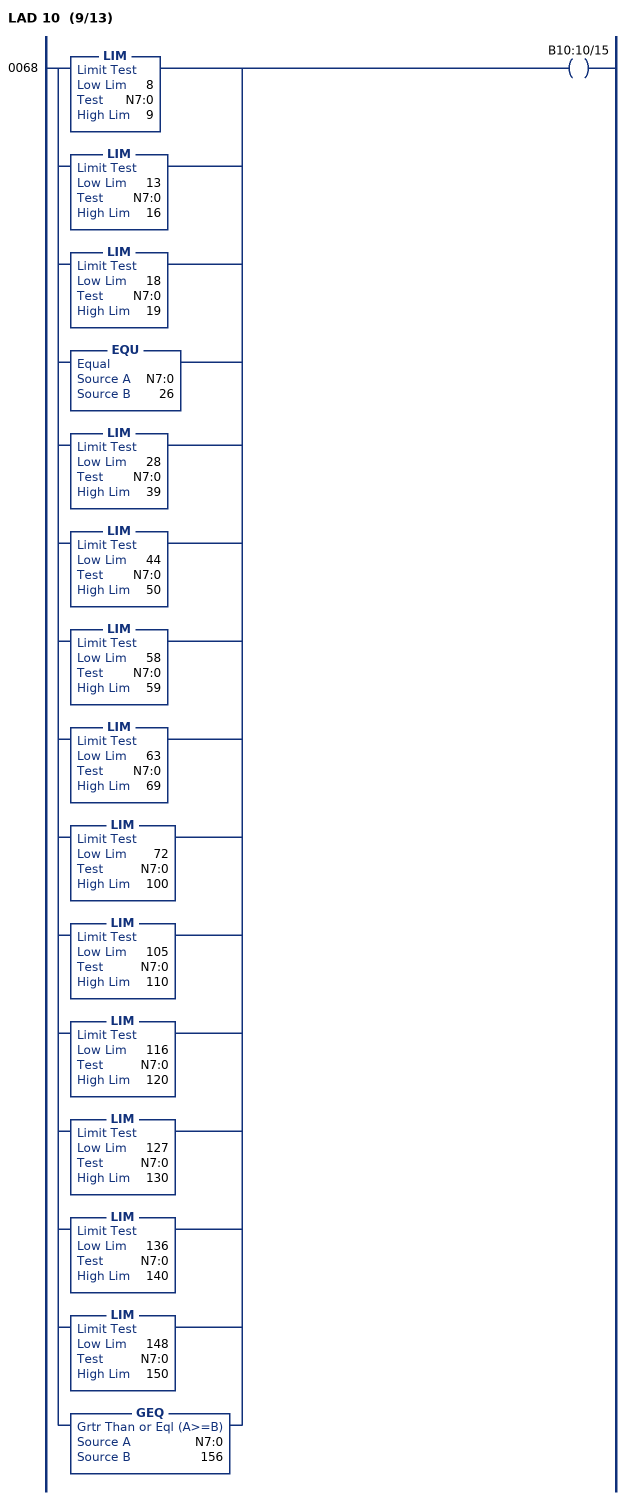
% Rung: 68 %
SOR BST LIM 8 N7:0 9 NXB LIM 13 N7:0 16 NXB LIM 18 N7:0 19 NXB EQU N7:0 26 NXB LIM 28 N7:0 39 NXB LIM 44 N7:0 50 NXB LIM 58 N7:0 59 NXB LIM 63 N7:0 69 NXB LIM 72 N7:0 100 NXB LIM 105 N7:0 110 NXB LIM 116 N7:0 120 NXB LIM 127 N7:0 130 NXB LIM 136 N7:0 140 NXB LIM 148 N7:0 150 NXB GEQ N7:0 156 BND OTE B10:10/15 EOR

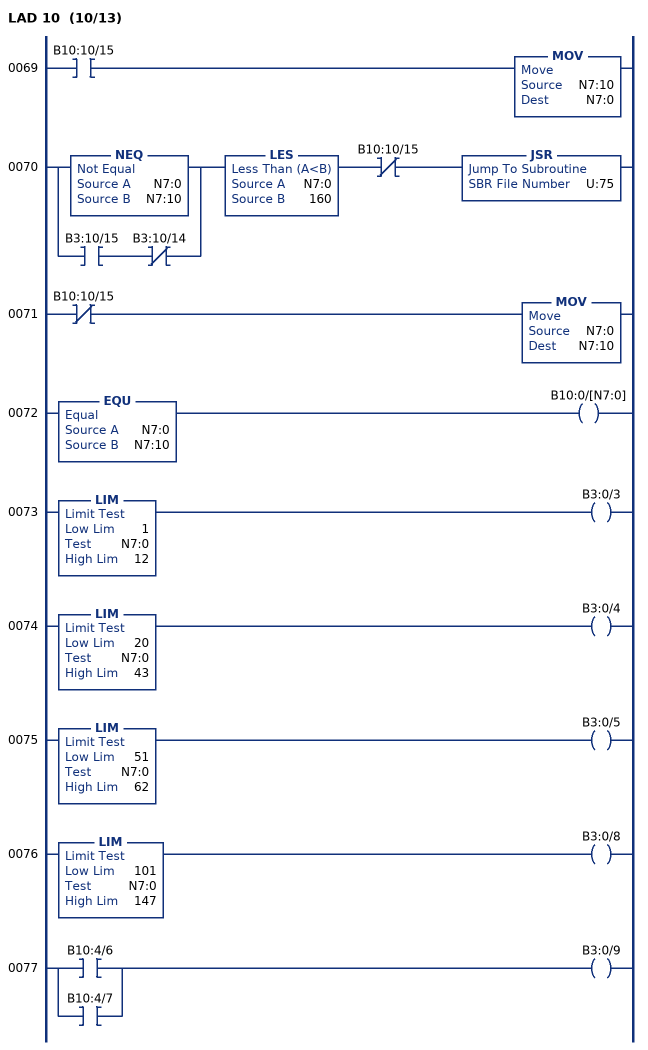
% Rung: 69 %
SOR XIC B10:10/15 MOV N7:10 N7:0 EOR
% Rung: 70 %
SOR BST NEQ N7:0 N7:10 NXB XIC B3:10/15 XIO B3:10/14 BND LES N7:0 160 XIO B10:10/15 JSR U:75 EOR
% Rung: 71 %
SOR XIO B10:10/15 MOV N7:0 N7:10 EOR
% Rung: 72 %
SOR EQU N7:0 N7:10 OTE B10:0/[N7:0] EOR
% Rung: 73 %
SOR LIM 1 N7:0 12 OTE B3:0/3 EOR
% Rung: 74 %
SOR LIM 20 N7:0 43 OTE B3:0/4 EOR
% Rung: 75 %
SOR LIM 51 N7:0 62 OTE B3:0/5 EOR
% Rung: 76 %
SOR LIM 101 N7:0 147 OTE B3:0/8 EOR
% Rung: 77 %
SOR BST XIC B10:4/6 NXB XIC B10:4/7 BND OTE B3:0/9 EOR

